// SIMATIC S7-200 project (STEP 7-Micro/WIN), CPU 222 CN REL 02.01

SYMBOL_TABLE 符号表
甲自动              I1.0     // 甲秤投入自动
乙自动              I1.1     // 乙秤投入自动
甲运行              I1.2     // 甲秤称量控制器送电运行
乙运行              I1.3     // 乙秤称量控制器送电运行
甲不足              I1.4     // 甲秤称量控制器显示不足
乙不足              I1.5     // 乙秤称量控制器显示不足
甲过量              I1.6     // 甲秤称量控制器显示过量
乙过量              I1.7     // 乙秤称量控制器显示过量
甲快加指示            I0.0     // 甲秤快加指示
甲慢加指示            I0.1     // 甲秤慢加指示
乙快加指示            I0.3     // 乙秤快加指示
乙慢加指示            I0.4     // 乙秤慢加指示
夹袋按钮             I0.6     // 夹袋指示
松袋按钮             I0.7     // 松袋指示
快加甲              Q0.0     // 甲秤快加动作
慢加甲              Q0.1     // 甲秤慢加动作
放料甲              Q0.2     // 甲秤放料动作
快加乙              Q0.3     // 乙秤快加动作
慢加乙              Q0.4     // 乙秤慢加动作
放料乙              Q0.5     // 乙秤放料动作
夹袋               Q1.0     // 夹袋动作，自动则持续n秒，手动须按松袋按钮
计数脉冲             Q1.1     // 送出计数脉冲
不足               Q1.2     // 甲秤或乙秤不足，电亮不足指示灯
过量               Q1.3     // 甲秤或乙秤过量，点亮过量指示灯
甲秤自动运行           M0.0     // 甲秤开关投入自动，称量控制器上电
乙秤自动运行           M0.1     // 乙秤开关投入自动，称量控制器上电
甲秤可以放料           M0.2     // 甲秤具备放料条件
乙秤可以放料           M0.3     // 乙秤具备放料条件
要求夹袋             M0.4     // 要求夹袋
要求松袋甲            M0.5     // 要求松袋甲
放料次数             M0.6     // 两秤放料次数
要求松袋乙            M0.7     // 要求松袋乙
输出脉冲             M1.0     // 输出脉冲
甲秤不得快慢加          M1.1     // 甲秤放料1.5s内不得快加慢加
乙秤不得快慢加          M1.2     // 乙秤放料1.5s内不得快加慢加
乙不准放料            M1.3     // 甲自动切换到手动期间乙不准放料
甲不准放料            M1.4     // 乙自动切换到手动期间甲不准放料
甲秤放料             M1.5     // 甲秤放料
乙秤放料             M1.6     // 乙秤放料
甲放料时间            T33      // 1s
甲松袋时间            T34      // 1.2s
乙放料时间            T35      // 1s
乙松袋时间            T36      // 1.2s
夹袋时间             T37      // 1s
计数宽度             T38      // 计数脉冲宽度0.5s
甲秤禁加料时间          T39      // 甲秤放料后到快慢加动作1.5s
乙秤禁加料时间          T40      // 乙秤放料后到快慢加动作1.5s
甲加到放料时间          T41      // 甲秤慢加完0.3s才能放料
乙加到放料时间          T42      // 乙秤慢加完0.3s才能放料
乙不准放料时间          T97      // 甲自动切换手动期间乙不准放料
甲不准放料时间          T98      // 乙自动切换手动期间甲不准放料
复合肥报数低           C0
复合肥报数高           C1
状态字              VW130
包数               VD30     // 复合肥包数
END_SYMBOL_TABLE

ORGANIZATION_BLOCK 程序块:OB1
TITLE=~~~项目
// 复合肥包装秤的控制程序。
// ~~~设备信息
// 系统控制的物理设备包括甲秤、乙秤、夹袋装置、松袋装置、指示灯和按钮。
// ~~~执行流程
// 甲秤通过自动运行控制加料，乙秤通过自动运行控制加料，两秤放料条件互斥实现交替工作，确保生产线连续运行。
// 操作员通过自动开关将甲秤和乙秤切换至自动模式，运行指示确认控制器已上电并准备就绪。
// 加料过程由快加指示和慢加指示触发快加输出和慢加输出。
// 加料仅在可以放料标志未置位且不得快慢加标志未置位时执行，避免与放料冲突。
// 甲秤完成加料后，系统检查快加指示、慢加指示、加到放料时间定时器和夹袋时间定时器是否满足条件，确保加料稳定且夹袋就位。
// 若乙秤可以放料标志未置位，甲秤可以放料标志置位。
// 在要求夹袋标志置位时，甲秤放料标志置位并启动放料时间定时器持续1秒，随后触发放料输出。
// 甲秤放料时，不得快慢加标志置位，随后通过禁加料时间定时器持续1.5秒，最终复位以释放禁加料状态，确保放料过程不受干扰。
// 乙秤放料标志置位并启动放料时间定时器，随后触发放料输出。
// 夹袋按钮触发要求夹袋标志置位，随后夹袋输出置位并持续1秒。
// 在设置甲秤和乙秤可以放料时，要求松袋标志不得置位，确保夹袋完成前不松袋。
// 松袋动作在放料时间定时器到时或松袋按钮被按下时触发，要求松袋标志置位并启动松袋时间定时器持续1.2秒，确保放料后安全松开袋子。
// 
BEGIN
Network 1
// 网络注解  I1.0---甲自动
LD     甲自动:I1.0
A      甲运行:I1.2
=      甲秤自动运行:M0.0
?000
Network 2
// 网络注解  I1.1---乙自动
LD     乙自动:I1.1
A      乙运行:I1.3
=      乙秤自动运行:M0.1
Network 3
// 网络注解  I1.4、I1.5---不足
LD     甲不足:I1.4
O      乙不足:I1.5
=      不足:Q1.2
Network 4
// 网络注解  I1.6、I1.7---过量
LD     甲过量:I1.6
O      乙过量:I1.7
=      过量:Q1.3
Network 5
// 甲秤    大小弧门开
LD     甲秤自动运行:M0.0
AN     甲秤可以放料:M0.2
AN     甲快加指示:I0.0
AN     甲秤不得快慢加:M1.1
=      快加甲:Q0.0
Network 6
// 甲秤    小弧门开
LD     甲秤自动运行:M0.0
AN     甲秤可以放料:M0.2
AN     甲慢加指示:I0.1
AN     甲秤不得快慢加:M1.1
=      慢加甲:Q0.1
Network 7
LD     甲慢加指示:I0.1
TON    甲加到放料时间:T41, 3
Network 8
LD     夹袋按钮:I0.6
O      要求夹袋:M0.4
AN     松袋按钮:I0.7
AN     甲松袋时间:T34
AN     乙松袋时间:T36
=      要求夹袋:M0.4
Network 9
// 夹袋
LD     要求夹袋:M0.4
=      夹袋:Q1.0
TON    夹袋时间:T37, 10
Network 10
// 甲秤    可以放料
LD     甲秤自动运行:M0.0
LD     甲快加指示:I0.0
A      甲慢加指示:I0.1
A      甲加到放料时间:T41
A      夹袋时间:T37
O      甲秤可以放料:M0.2
ALD
AN     乙秤可以放料:M0.3
AN     要求松袋甲:M0.5
AN     要求松袋乙:M0.7
=      甲秤可以放料:M0.2
Network 11
//     没有使用
LD     甲不准放料时间:T98
O      乙秤自动运行:M0.1
R      甲不准放料:M1.4, 1
Network 12
// 甲秤    放料
LD     要求夹袋:M0.4
A      甲秤可以放料:M0.2
O      甲秤放料:M1.5
AN     要求松袋甲:M0.5
AN     乙秤放料:M1.6
=      甲秤放料:M1.5
TON    甲放料时间:T33, 100
S      甲秤不得快慢加:M1.1, 1
Network 13
LD     甲秤放料:M1.5
=      放料甲:Q0.2
Network 14
LD     甲秤不得快慢加:M1.1
TON    甲秤禁加料时间:T39, 15
Network 15
LD     甲秤禁加料时间:T39
R      甲秤不得快慢加:M1.1, 1
Network 16
// 松袋
LD     甲放料时间:T33
O      松袋按钮:I0.7
O      要求松袋甲:M0.5
AN     甲松袋时间:T34
=      要求松袋甲:M0.5
R      甲放料时间:T33, 1
R      放料甲:Q0.2, 1
TON    甲松袋时间:T34, 120
Network 17
// 乙秤    大小弧门开
LD     乙秤自动运行:M0.1
AN     乙秤可以放料:M0.3
AN     乙快加指示:I0.3
AN     乙秤不得快慢加:M1.2
=      快加乙:Q0.3
Network 18
// 乙秤    小弧门开
LD     乙秤自动运行:M0.1
AN     乙秤可以放料:M0.3
AN     乙慢加指示:I0.4
AN     乙秤不得快慢加:M1.2
=      慢加乙:Q0.4
Network 19
LD     乙慢加指示:I0.4
TON    乙加到放料时间:T42, 3
Network 20
// 乙秤    放料
LD     乙秤自动运行:M0.1
LD     乙快加指示:I0.3
A      乙慢加指示:I0.4
A      乙加到放料时间:T42
A      夹袋时间:T37
O      乙秤可以放料:M0.3
ALD
AN     甲秤可以放料:M0.2
AN     要求松袋甲:M0.5
AN     要求松袋乙:M0.7
=      乙秤可以放料:M0.3
Network 21
LD     要求夹袋:M0.4
A      乙秤可以放料:M0.3
O      乙秤放料:M1.6
AN     要求松袋乙:M0.7
AN     甲秤放料:M1.5
=      乙秤放料:M1.6
TON    乙放料时间:T35, 100
S      乙秤不得快慢加:M1.2, 1
Network 22
LD     乙秤放料:M1.6
=      放料乙:Q0.5
Network 23
// 松袋
LD     乙放料时间:T35
O      松袋按钮:I0.7
O      要求松袋乙:M0.7
AN     乙松袋时间:T36
=      要求松袋乙:M0.7
R      乙放料时间:T35, 1
R      放料乙:Q0.5, 1
TON    乙松袋时间:T36, 120
Network 24
LD     乙秤不得快慢加:M1.2
TON    乙秤禁加料时间:T40, 15
Network 25
LD     乙秤禁加料时间:T40
R      乙秤不得快慢加:M1.2, 1
Network 26
// 放料次数
LD     甲秤自动运行:M0.0
A      放料甲:Q0.2
LD     乙秤自动运行:M0.1
A      放料乙:Q0.5
OLD
=      放料次数:M0.6
Network 27
// 放料次数    1秒50%脉冲
LD     放料次数:M0.6
EU
S      输出脉冲:M1.0, 1
Network 28
LD     输出脉冲:M1.0
TON    计数宽度:T38, 5
Network 29
LD     计数宽度:T38
R      输出脉冲:M1.0, 1
Network 30
// 放料次数    1秒50%脉冲    输出到计数器
LD     输出脉冲:M1.0
=      计数脉冲:Q1.1
Network 31
// T2复位
LD     甲松袋时间:T34
O      乙松袋时间:T36
R      夹袋:Q1.0, 1
Network 32
LD     SM0.0
CALL   SBR_0:SBR0
END_ORGANIZATION_BLOCK

SUBROUTINE_BLOCK SBR_0:SBR0
TITLE=子程序注释
BEGIN
Network 1
// VB100 ~ VB103    存放复合肥包数
LD     输出脉冲:M1.0
LDD>=  包数:VD30, 32767
CTU    复合肥报数低:C0, 0
Network 2
LDD>=  包数:VD30, 32767
LD     SM0.1
CTU    复合肥报数高:C1, 0
Network 3
LDD>=  包数:VD30, 32767
R      复合肥报数低:C0, 1
Network 4 // 网络标题
// 网络注释
LD     甲秤自动运行:M0.0
=      V130.0
Network 5
LD     乙秤自动运行:M0.1
=      V130.1
Network 6
LD     快加甲:Q0.0
=      V130.2
Network 7
LD     慢加甲:Q0.1
=      V130.3
Network 8
LD     放料甲:Q0.2
=      V130.4
Network 9
LD     快加乙:Q0.3
=      V130.5
Network 10
LD     慢加乙:Q0.4
=      V130.6
Network 11
LD     放料乙:Q0.5
=      V130.7
Network 12
LD     夹袋:Q1.0
=      V131.0
Network 13
LD     不足:Q1.2
=      V131.1
Network 14
LD     过量:Q1.3
=      V131.2
Network 15
LD     SM0.0
MOVW   甲放料时间:T33, VW50
MOVW   甲松袋时间:T34, VW70
MOVW   乙放料时间:T35, VW90
MOVW   乙松袋时间:T36, VW100
END_SUBROUTINE_BLOCK

DATA_BLOCK_TAB TD_DATA_0
BEGIN
VB0      'TD'
VB2      16#60               //设置‘语言’为 中文，设置‘更新速率’为 尽可能快
VB3      16#90               //设置显示为 20 字符模式； ENTER 键 V3.1；‘向上’键 V3.2；‘向下’键 V3.3；
VB4      6                   //设置信息条数
VB5      16#0                //设置功能键对应位为 M0.0 - M0.7，F 键已配置为置位 M 位
VW6      24                  //将信息起始地址设为 VB24
VW8      14                  //将信息使能位起始地址设为 VW14
VW10     65535               //全局密码（如使能）
VW12     256                 //字符集 = 简体中文
//MESSAGE 1
//信息使能位 V14.7
VB24     '包数'
VB28     16#11               //编辑通知 V28.2；确认通知 V28.1；无密码；
VB29     16#40               //无符号双字； 小数点右侧保留 0 位小数；
         包数, 16#0            //嵌入数据：将数据传送到此处显示。
VB34     '          '
//MESSAGE 2
//信息使能位 V14.6
VB44     ' T1 '
VB48     16#11               //编辑通知 V48.2；确认通知 V48.1；无密码；
VB49     16#10               //有符号字； 小数点右侧保留 0 位小数；
VW50     16#0                //嵌入数据：将数据传送到此处显示。
VB52     '            '
//MESSAGE 3
//信息使能位 V14.5
VB64     ' T2 '
VB68     16#11               //编辑通知 V68.2；确认通知 V68.1；无密码；
VB69     16#10               //有符号字； 小数点右侧保留 0 位小数；
VW70     16#0                //嵌入数据：将数据传送到此处显示。
VB72     '            '
//MESSAGE 4
//信息使能位 V14.4
VB84     ' T3 '
VB88     16#11               //编辑通知 V88.2；确认通知 V88.1；无密码；
VB89     16#10               //有符号字； 小数点右侧保留 0 位小数；
VW90     16#0                //嵌入数据：将数据传送到此处显示。
VB92     '            '
//MESSAGE 5
//信息使能位 V14.3
VB104    ' T4 '
VB108    16#11               //编辑通知 V108.2；确认通知 V108.1；无密码；
VB109    16#10               //有符号字； 小数点右侧保留 0 位小数；
VW110    16#0                //嵌入数据：将数据传送到此处显示。
VB112    '            '
//MESSAGE 6
//信息使能位 V14.2
VB124    '状态'
VB128    16#11               //编辑通知 V128.2；确认通知 V128.1；无密码；
VB129    16#30               //无符号字； 小数点右侧保留 0 位小数；
         状态字, 16#0           //嵌入数据：将数据传送到此处显示。
VB132    '            '
//END TD200_BLOCK ------------------------------
//数据页注释
//按 F1 键获取帮助和示范数据页
END_DATA_BLOCK_TAB
